// TIA Portal project "Siemens_V17" (V17)

(* hardware
DEVICE "S7-1200-Station_1"  S7-1200 Station
   slot 0: "Baugruppenträger_0"  S7-1200 Rack  Rack  V1.0
   slot 1: "Asset-Interface"  CPU 1211C DC/DC/DC  6ES7 211-1AE40-0XB0  V4.4
*)

// ===== PLC "Asset-Interface"  CPU 1211C DC/DC/DC =====

VAR_GLOBAL   // PLC tag table "Standard-Variablentabelle"
   "System_Byte" AT %MB1 : Byte;
   "FirstScan" AT %M1.0 : Bool;
   "DiagStatusUpdate" AT %M1.1 : Bool;
   "AlwaysTRUE" AT %M1.2 : Bool;
   "AlwaysFALSE" AT %M1.3 : Bool;
   "System_Byte(1)" AT %MB1 : Byte;
   "Clock_Byte" AT %MB0 : Byte;
   "Clock_10Hz" AT %M0.0 : Bool;
   "Clock_5Hz" AT %M0.1 : Bool;
   "Clock_2.5Hz" AT %M0.2 : Bool;
   "Clock_2Hz" AT %M0.3 : Bool;
   "Clock_1.25Hz" AT %M0.4 : Bool;
   "Clock_1Hz" AT %M0.5 : Bool;
   "Clock_0.625Hz" AT %M0.6 : Bool;
   "Clock_0.5Hz" AT %M0.7 : Bool;
END_VAR

TYPE "LivaAssetDataV1"
   STRUCT
      LivaDataId : Array[0..3] of Char;
      ModelId : UInt := 16#201;   // ID of model data structure = AssetValues
      Length : UInt := 27;   // Anzahl der folgenden Register
      AssetId : UInt := 0;   // Eindeutige ID des Assets aus der Konfiguration
      OperatingState : UInt := 4;   // Betriebszustand des Assets
      AlarmState : Array[0..63] of Bool;   // Meldungen / Alarme des Assets
      ActiveConsumption : UDInt := 0;   // [W] Momentane Leistungsaufnahme (laden / Verbrauch
      ActiveProduction : UDInt := 0;   // [W] Momentane Leistungsabgabe (entladen / Einspeisung)
      ReactiveCapacitive : UDInt := 0;   // [var] Momentane kapazitive Blindleistung
      ReactiveInductive : UDInt := 0;   // [var] Momentane induktive Blindleistung
      Temperature : Int := 0;   // [1/10 °] Interne Maximaltemperatur
      CapacityLevel : UDInt := 0;   // [Wh] Effektiver Ladezustand (SoC) des Assets
      ControlState : UInt := 0;   // Steuerungszustand
      ControlActivation : UInt := 0;   // Steuerungsvorgabe
      SetActiveConsume : UDInt := 0;   // [W] Vorgabe der Leistungsaufnahme (laden / Verbrauch)
      SetActiveProduce : UDInt := 0;   // [W] Vorgabe der Leistungsabgabe (entladen / Einspeisung)
      SetReactiveCapacitive : UDInt := 0;   // [var] Vorgabe der kapazitiven Blindleistung
      SetReactiveInductive : UDInt := 0;   // [var] Vorgabe der induktiven Blindleistung
   END_STRUCT;
   // LivaDataId[0] := CHAR#'L';
   // LivaDataId[1] := CHAR#'I';
   // LivaDataId[2] := CHAR#'V';
   // LivaDataId[3] := CHAR#'A';
END_TYPE

DATA_BLOCK "AssetModbusServer_DB"   // DB1
{ S7_Optimized_Access := 'TRUE' }
VERSION : 0.1
// stored: InstanceOfName AssetModbusServer
"AssetModbusServer"
BEGIN
END_DATA_BLOCK

DATA_BLOCK "WwwState"   // DB2
{ S7_Optimized_Access := 'TRUE' }
VERSION : 0.1
   VAR
      "WWW-Status" : Word;
   END_VAR
BEGIN
END_DATA_BLOCK

DATA_BLOCK "Asset-DB"   // DB3
{ S7_Optimized_Access := 'FALSE' }
VERSION : 0.1
   VAR
      AssetData : Array[0..9] of "LivaAssetDataV1";
   END_VAR
BEGIN
END_DATA_BLOCK

FUNCTION_BLOCK "AssetModbusServer"   // FB1, SCL
{ S7_Optimized_Access := 'TRUE' }
VERSION : 0.1
   VAR_INPUT
      disconnect : Bool;
   END_VAR
   VAR_OUTPUT
      ndr : Bool;
      dataRead : Bool;
      error : Bool;
      status : Word;
   END_VAR
   VAR
      MbServer : MB_SERVER;
      connectParamServer : TCON_IP_v4;
      ModbusState : Word;
   END_VAR
   // connectParamServer.InterfaceId := 64;
   // connectParamServer.ID := 1;
   // connectParamServer.LocalPort := 502;
   // connectParamServer.RemoteAddress.ADDR[1] := 0;
   // connectParamServer.RemoteAddress.ADDR[2] := 0;
   // connectParamServer.RemoteAddress.ADDR[3] := 0;
   // connectParamServer.RemoteAddress.ADDR[4] := 0;
BEGIN

   #MbServer(DISCONNECT := #disconnect,
             NDR => #ndr,
             DR => #dataRead,
             ERROR => #error,
             STATUS => #status,
             MB_HOLD_REG := "Asset-DB".AssetData,
             CONNECT := #connectParamServer);
END_FUNCTION_BLOCK

ORGANIZATION_BLOCK "Main"   // OB1, LAD, ProgramCycle
TITLE = "Main Program Sweep (Cycle)"
{ S7_Optimized_Access := 'TRUE' }
VERSION : 0.1
   VAR_INPUT
      Initial_Call : Bool;   // Initial call of this OB
      Remanence : Bool;   // =True, if remanent data are available
   END_VAR
BEGIN

REGION Network 1
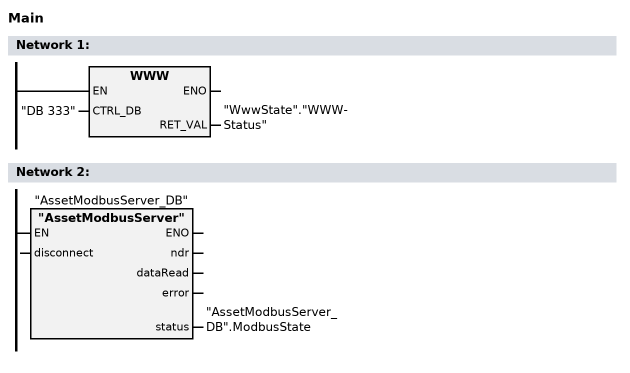
   "WwwState"."WWW-Status" := WWW(CTRL_DB := "DB 333");
END_REGION

REGION Network 2
   RUNG wire#powerrail
      "AssetModbusServer_DB"(disconnect :=, ndr =>, dataRead =>, error =>, status => "AssetModbusServer_DB".ModbusState)
   END_RUNG
   // the same network as SCL:
   "AssetModbusServer_DB"(status => "AssetModbusServer_DB".ModbusState);   // "AssetModbusServer"
END_REGION
END_ORGANIZATION_BLOCK